// TIA Portal V20 export
FUNCTION "Block_1" : Void   // FC1, FBD
{ S7_Optimized_Access := 'TRUE' }
// stored: SetENOAutomatically false
BEGIN
END_FUNCTION
